// TwinCAT 3 PLC project plc
// ProgramVersion: 3.1.4024.0
// libraries:
//   Tc2_Standard, * (Beckhoff Automation GmbH)
//   Tc2_System, * (Beckhoff Automation GmbH)
//   Tc3_Module, * (Beckhoff Automation GmbH)
// project tree:
//   DUTs/ Axis_Command.TcDUT, Axis_Status.TcDUT
//   / PlcTask.TcTTO
//   POUs/ MAIN.TcPOU
// real-time tasks:
//   TASK PlcTask: cycle T#1ms, priority 4, ADS port 350
//   TASK PlcTask1: cycle T#2ms, priority 6, ADS port 351
// I/O:
//   DEVICE Device 2 (EtherCAT), AmsNetId 169.254.115.184.3.1
//     Box 2 (EX1616DN) [EX1616DN]
//       modules: Module 1 (SX1616DN)
//     p1 [MCDLN35BE]
//     j1 [MDDLN55BE]
//     j2 [MDDLN55BE]
//     j3 [MDDLN55BE]
//     j4 [MCDLN35BE]
//     j5 [MCDLN35BE]
//     j6 [MBDLN25BE]
//   DEVICE Device 4 (EtherCAT) (disabled), AmsNetId 172.16.9.47.5.1
//     zhua1 [ZeroErr Driver]
//     zhua2 [ZeroErr Driver]
//     kuaisubanshou1 [ZeroErr Driver] (disabled)
//     kuaisubanshou2 [ZeroErr Driver] (disabled)
//     kuaisubanshouqianjin [ZeroErr Driver] (disabled)
//   DEVICE Device 1 (EtherCAT) (disabled), AmsNetId 172.16.9.47.2.1
//     Drive 5 (ZeroErr Driver) [ZeroErr Driver]
// variable links:
//   plc2/plc2 Instance <-> Device 1 (EtherCAT)/Drive 5 (ZeroErr Driver)
//     PlcTask Inputs/MAIN.TW_STATUS/POSITION <-> Transmit PDO mapping 2/Position actual value
//     PlcTask Inputs/MAIN.TW_STATUS/STATUS_WORD <-> Transmit PDO mapping 2/Status word
//     PlcTask Inputs/MAIN.TW_STATUS/TORQUE_VALUE <-> Transmit PDO mapping 2/Torque actual value
//     PlcTask Outputs/MAIN.TW_COMMAND/CONTROL_WORD <-> Receive PDO mapping 8/Controlword
//     PlcTask Outputs/MAIN.TW_COMMAND/MAX_MOTOR_SPEED <-> Receive PDO mapping 8/Max motor speed
//     PlcTask Outputs/MAIN.TW_COMMAND/MODE_OF_OPERATION <-> Receive PDO mapping 8/Modes of operation
//     PlcTask Outputs/MAIN.TW_COMMAND/TARGET_TORQUE <-> Receive PDO mapping 8/Target torque
//   plc2/plc2 Instance <-> Device 4 (EtherCAT)/kuaisubanshou1
//     PlcTask Inputs/MAIN.T_Axis_3_STATUS/POSITION <-> Transmit PDO mapping 2/Position actual value
//     PlcTask Inputs/MAIN.T_Axis_3_STATUS/STATUS_WORD <-> Transmit PDO mapping 2/Status word
//     PlcTask Inputs/MAIN.T_Axis_3_STATUS/TORQUE_VALUE <-> Transmit PDO mapping 2/Torque actual value
//     PlcTask Outputs/MAIN.T_Axis_3_COMMAND/CONTROL_WORD <-> Receive PDO mapping 8/Controlword
//     PlcTask Outputs/MAIN.T_Axis_3_COMMAND/MAX_MOTOR_SPEED <-> Receive PDO mapping 8/Max motor speed
//     PlcTask Outputs/MAIN.T_Axis_3_COMMAND/MODE_OF_OPERATION <-> Receive PDO mapping 8/Modes of operation
//     PlcTask Outputs/MAIN.T_Axis_3_COMMAND/TARGET_TORQUE <-> Receive PDO mapping 8/Target torque
//   plc2/plc2 Instance <-> Device 4 (EtherCAT)/kuaisubanshou2
//     PlcTask Inputs/MAIN.T_Axis_4_STATUS/POSITION <-> Transmit PDO mapping 2/Position actual value
//     PlcTask Inputs/MAIN.T_Axis_4_STATUS/STATUS_WORD <-> Transmit PDO mapping 2/Status word
//     PlcTask Inputs/MAIN.T_Axis_4_STATUS/TORQUE_VALUE <-> Transmit PDO mapping 2/Torque actual value
//     PlcTask Outputs/MAIN.T_Axis_4_COMMAND/CONTROL_WORD <-> Receive PDO mapping 8/Controlword
//     PlcTask Outputs/MAIN.T_Axis_4_COMMAND/MAX_MOTOR_SPEED <-> Receive PDO mapping 8/Max motor speed
//     PlcTask Outputs/MAIN.T_Axis_4_COMMAND/MODE_OF_OPERATION <-> Receive PDO mapping 8/Modes of operation
//     PlcTask Outputs/MAIN.T_Axis_4_COMMAND/TARGET_TORQUE <-> Receive PDO mapping 8/Target torque
//   plc2/plc2 Instance <-> Device 4 (EtherCAT)/kuaisubanshouqianjin
//     PlcTask Inputs/MAIN.P_Axis_1_STATUS/POSITION_VALUE <-> Transmit PDO mapping 0/Position actual value
//     PlcTask Inputs/MAIN.P_Axis_1_STATUS/STATUS_WORD <-> Transmit PDO mapping 0/Status word
//     PlcTask Outputs/MAIN.P_Axis_1_COMMAND/CONTROL_WORD <-> Receive PDO mapping 7/Control word
//     PlcTask Outputs/MAIN.P_Axis_1_COMMAND/MODE_OF_OPERATION <-> Receive PDO mapping 7/Mode of operation
//     PlcTask Outputs/MAIN.P_Axis_1_COMMAND/TARGET_POSITION <-> Receive PDO mapping 7/Target Position
//   plc2/plc2 Instance <-> Device 4 (EtherCAT)/zhua1
//     PlcTask Inputs/MAIN.T_Axis_1_STATUS/POSITION <-> Transmit PDO mapping 2/Position actual value
//     PlcTask Inputs/MAIN.T_Axis_1_STATUS/STATUS_WORD <-> Transmit PDO mapping 2/Status word
//     PlcTask Inputs/MAIN.T_Axis_1_STATUS/TORQUE_VALUE <-> Transmit PDO mapping 2/Torque actual value
//     PlcTask Outputs/MAIN.T_Axis_1_COMMAND/CONTROL_WORD <-> Receive PDO mapping 8/Controlword
//     PlcTask Outputs/MAIN.T_Axis_1_COMMAND/MAX_MOTOR_SPEED <-> Receive PDO mapping 8/Max motor speed
//     PlcTask Outputs/MAIN.T_Axis_1_COMMAND/MODE_OF_OPERATION <-> Receive PDO mapping 8/Modes of operation
//     PlcTask Outputs/MAIN.T_Axis_1_COMMAND/TARGET_TORQUE <-> Receive PDO mapping 8/Target torque
//   plc2/plc2 Instance <-> Device 4 (EtherCAT)/zhua2
//     PlcTask Inputs/MAIN.T_Axis_2_STATUS/POSITION <-> Transmit PDO mapping 2/Position actual value
//     PlcTask Inputs/MAIN.T_Axis_2_STATUS/STATUS_WORD <-> Transmit PDO mapping 2/Status word
//     PlcTask Inputs/MAIN.T_Axis_2_STATUS/TORQUE_VALUE <-> Transmit PDO mapping 2/Torque actual value
//     PlcTask Outputs/MAIN.T_Axis_2_COMMAND/CONTROL_WORD <-> Receive PDO mapping 8/Controlword
//     PlcTask Outputs/MAIN.T_Axis_2_COMMAND/MAX_MOTOR_SPEED <-> Receive PDO mapping 8/Max motor speed
//     PlcTask Outputs/MAIN.T_Axis_2_COMMAND/MODE_OF_OPERATION <-> Receive PDO mapping 8/Modes of operation
//     PlcTask Outputs/MAIN.T_Axis_2_COMMAND/TARGET_TORQUE <-> Receive PDO mapping 8/Target torque
//   plc/plc Instance <-> Device 2 (EtherCAT)/Box 2 (EX1616DN)
//     PlcTask Outputs/MAIN.BREAK <-> Module 1 (SX1616DN)/Outputs/Digital16 OUT
//   plc/plc Instance <-> Device 2 (EtherCAT)/j1
//     PlcTask Inputs/MAIN.j1_status/Actual_Position <-> Transmit PDO mapping 1/Position actual value
//     PlcTask Inputs/MAIN.j1_status/Actual_Torque <-> Transmit PDO mapping 1/Torque actual value
//     PlcTask Inputs/MAIN.j1_status/Actual_Velocity <-> Transmit PDO mapping 1/Velocity actual value
//     PlcTask Inputs/MAIN.j1_status/Following_Err <-> Transmit PDO mapping 1/Following error actual value
//     PlcTask Inputs/MAIN.j1_status/Mode_of_Operation_disp <-> Transmit PDO mapping 1/Modes of operation display
//     PlcTask Inputs/MAIN.j1_status/status <-> Transmit PDO mapping 1/Statusword
//     PlcTask Outputs/MAIN.j1_acc <-> Receive PDO mapping 1/Profile acceleration
//     PlcTask Outputs/MAIN.j1_command/Control_Word <-> Receive PDO mapping 1/Controlword
//     PlcTask Outputs/MAIN.j1_command/Max_Motor_Speed <-> Receive PDO mapping 1/Max motor speed
//     PlcTask Outputs/MAIN.j1_command/Max_Torque <-> Receive PDO mapping 1/Max torque
//     PlcTask Outputs/MAIN.j1_command/Mode_of_Operation <-> Receive PDO mapping 1/Modes of operation
//     PlcTask Outputs/MAIN.j1_command/Profile_Velocity <-> Receive PDO mapping 1/Profile velocity
//     PlcTask Outputs/MAIN.j1_command/Target_Position <-> Receive PDO mapping 1/Target position
//     PlcTask Outputs/MAIN.j1_command/Target_Torque <-> Receive PDO mapping 1/Target torque
//     PlcTask Outputs/MAIN.j1_dacc <-> Receive PDO mapping 1/Profile deceleration
//   plc/plc Instance <-> Device 2 (EtherCAT)/j2
//     PlcTask Inputs/MAIN.j2_status/Actual_Position <-> Transmit PDO mapping 1/Position actual value
//     PlcTask Inputs/MAIN.j2_status/Actual_Torque <-> Transmit PDO mapping 1/Torque actual value
//     PlcTask Inputs/MAIN.j2_status/Actual_Velocity <-> Transmit PDO mapping 1/Velocity actual value
//     PlcTask Inputs/MAIN.j2_status/Following_Err <-> Transmit PDO mapping 1/Following error actual value
//     PlcTask Inputs/MAIN.j2_status/Mode_of_Operation_disp <-> Transmit PDO mapping 1/Modes of operation display
//     PlcTask Inputs/MAIN.j2_status/status <-> Transmit PDO mapping 1/Statusword
//     PlcTask Outputs/MAIN.j2_acc <-> Receive PDO mapping 1/Profile acceleration
//     PlcTask Outputs/MAIN.j2_command/Control_Word <-> Receive PDO mapping 1/Controlword
//     PlcTask Outputs/MAIN.j2_command/Max_Motor_Speed <-> Receive PDO mapping 1/Max motor speed
//     PlcTask Outputs/MAIN.j2_command/Max_Torque <-> Receive PDO mapping 1/Max torque
//     PlcTask Outputs/MAIN.j2_command/Mode_of_Operation <-> Receive PDO mapping 1/Modes of operation
//     PlcTask Outputs/MAIN.j2_command/Profile_Velocity <-> Receive PDO mapping 1/Profile velocity
//     PlcTask Outputs/MAIN.j2_command/Target_Position <-> Receive PDO mapping 1/Target position
//     PlcTask Outputs/MAIN.j2_command/Target_Torque <-> Receive PDO mapping 1/Target torque
//     PlcTask Outputs/MAIN.j2_dacc <-> Receive PDO mapping 1/Profile deceleration
//   plc/plc Instance <-> Device 2 (EtherCAT)/j3
//     PlcTask Inputs/MAIN.j3_status/Actual_Position <-> Transmit PDO mapping 1/Position actual value
//     PlcTask Inputs/MAIN.j3_status/Actual_Torque <-> Transmit PDO mapping 1/Torque actual value
//     PlcTask Inputs/MAIN.j3_status/Actual_Velocity <-> Transmit PDO mapping 1/Velocity actual value
//     PlcTask Inputs/MAIN.j3_status/Following_Err <-> Transmit PDO mapping 1/Following error actual value
//     PlcTask Inputs/MAIN.j3_status/Mode_of_Operation_disp <-> Transmit PDO mapping 1/Modes of operation display
//     PlcTask Inputs/MAIN.j3_status/status <-> Transmit PDO mapping 1/Statusword
//     PlcTask Outputs/MAIN.j3_acc <-> Receive PDO mapping 1/Profile acceleration
//     PlcTask Outputs/MAIN.j3_command/Control_Word <-> Receive PDO mapping 1/Controlword
//     PlcTask Outputs/MAIN.j3_command/Max_Motor_Speed <-> Receive PDO mapping 1/Max motor speed
//     PlcTask Outputs/MAIN.j3_command/Max_Torque <-> Receive PDO mapping 1/Max torque
//     PlcTask Outputs/MAIN.j3_command/Mode_of_Operation <-> Receive PDO mapping 1/Modes of operation
//     PlcTask Outputs/MAIN.j3_command/Profile_Velocity <-> Receive PDO mapping 1/Profile velocity
//     PlcTask Outputs/MAIN.j3_command/Target_Position <-> Receive PDO mapping 1/Target position
//     PlcTask Outputs/MAIN.j3_command/Target_Torque <-> Receive PDO mapping 1/Target torque
//     PlcTask Outputs/MAIN.j3_dacc <-> Receive PDO mapping 1/Profile deceleration
//   plc/plc Instance <-> Device 2 (EtherCAT)/j4
//     PlcTask Inputs/MAIN.j4_status/Actual_Position <-> Transmit PDO mapping 1/Position actual value
//     PlcTask Inputs/MAIN.j4_status/Actual_Torque <-> Transmit PDO mapping 1/Torque actual value
//     PlcTask Inputs/MAIN.j4_status/Actual_Velocity <-> Transmit PDO mapping 1/Velocity actual value
//     PlcTask Inputs/MAIN.j4_status/Following_Err <-> Transmit PDO mapping 1/Following error actual value
//     PlcTask Inputs/MAIN.j4_status/Mode_of_Operation_disp <-> Transmit PDO mapping 1/Modes of operation display
//     PlcTask Inputs/MAIN.j4_status/status <-> Transmit PDO mapping 1/Statusword
//     PlcTask Outputs/MAIN.j4_acc <-> Receive PDO mapping 1/Profile acceleration
//     PlcTask Outputs/MAIN.j4_command/Control_Word <-> Receive PDO mapping 1/Controlword
//     PlcTask Outputs/MAIN.j4_command/Max_Motor_Speed <-> Receive PDO mapping 1/Max motor speed
//     PlcTask Outputs/MAIN.j4_command/Max_Torque <-> Receive PDO mapping 1/Max torque
//     PlcTask Outputs/MAIN.j4_command/Mode_of_Operation <-> Receive PDO mapping 1/Modes of operation
//     PlcTask Outputs/MAIN.j4_command/Profile_Velocity <-> Receive PDO mapping 1/Profile velocity
//     PlcTask Outputs/MAIN.j4_command/Target_Position <-> Receive PDO mapping 1/Target position
//     PlcTask Outputs/MAIN.j4_command/Target_Torque <-> Receive PDO mapping 1/Target torque
//     PlcTask Outputs/MAIN.j4_dacc <-> Receive PDO mapping 1/Profile deceleration
//   plc/plc Instance <-> Device 2 (EtherCAT)/j5
//     PlcTask Inputs/MAIN.j5_status/Actual_Position <-> Transmit PDO mapping 1/Position actual value
//     PlcTask Inputs/MAIN.j5_status/Actual_Torque <-> Transmit PDO mapping 1/Torque actual value
//     PlcTask Inputs/MAIN.j5_status/Actual_Velocity <-> Transmit PDO mapping 1/Velocity actual value
//     PlcTask Inputs/MAIN.j5_status/Following_Err <-> Transmit PDO mapping 1/Following error actual value
//     PlcTask Inputs/MAIN.j5_status/Mode_of_Operation_disp <-> Transmit PDO mapping 1/Modes of operation display
//     PlcTask Inputs/MAIN.j5_status/status <-> Transmit PDO mapping 1/Statusword
//     PlcTask Outputs/MAIN.j5_acc <-> Receive PDO mapping 1/Profile acceleration
//     PlcTask Outputs/MAIN.j5_command/Control_Word <-> Receive PDO mapping 1/Controlword
//     PlcTask Outputs/MAIN.j5_command/Max_Motor_Speed <-> Receive PDO mapping 1/Max motor speed
//     PlcTask Outputs/MAIN.j5_command/Max_Torque <-> Receive PDO mapping 1/Max torque
//     PlcTask Outputs/MAIN.j5_command/Mode_of_Operation <-> Receive PDO mapping 1/Modes of operation
//     PlcTask Outputs/MAIN.j5_command/Profile_Velocity <-> Receive PDO mapping 1/Profile velocity
//     PlcTask Outputs/MAIN.j5_command/Target_Position <-> Receive PDO mapping 1/Target position
//     PlcTask Outputs/MAIN.j5_command/Target_Torque <-> Receive PDO mapping 1/Target torque
//     PlcTask Outputs/MAIN.j5_dacc <-> Receive PDO mapping 1/Profile deceleration
//   plc/plc Instance <-> Device 2 (EtherCAT)/j6
//     PlcTask Inputs/MAIN.j6_status/Actual_Position <-> Transmit PDO mapping 1/Position actual value
//     PlcTask Inputs/MAIN.j6_status/Actual_Torque <-> Transmit PDO mapping 1/Torque actual value
//     PlcTask Inputs/MAIN.j6_status/Actual_Velocity <-> Transmit PDO mapping 1/Velocity actual value
//     PlcTask Inputs/MAIN.j6_status/Following_Err <-> Transmit PDO mapping 1/Following error actual value
//     PlcTask Inputs/MAIN.j6_status/Mode_of_Operation_disp <-> Transmit PDO mapping 1/Modes of operation display
//     PlcTask Inputs/MAIN.j6_status/status <-> Transmit PDO mapping 1/Statusword
//     PlcTask Outputs/MAIN.j6_acc <-> Receive PDO mapping 1/Profile acceleration
//     PlcTask Outputs/MAIN.j6_command/Control_Word <-> Receive PDO mapping 1/Controlword
//     PlcTask Outputs/MAIN.j6_command/Max_Motor_Speed <-> Receive PDO mapping 1/Max motor speed
//     PlcTask Outputs/MAIN.j6_command/Max_Torque <-> Receive PDO mapping 1/Max torque
//     PlcTask Outputs/MAIN.j6_command/Mode_of_Operation <-> Receive PDO mapping 1/Modes of operation
//     PlcTask Outputs/MAIN.j6_command/Profile_Velocity <-> Receive PDO mapping 1/Profile velocity
//     PlcTask Outputs/MAIN.j6_command/Target_Position <-> Receive PDO mapping 1/Target position
//     PlcTask Outputs/MAIN.j6_command/Target_Torque <-> Receive PDO mapping 1/Target torque
//     PlcTask Outputs/MAIN.j6_dacc <-> Receive PDO mapping 1/Profile deceleration
//   plc/plc Instance <-> Device 2 (EtherCAT)/p1
//     PlcTask Inputs/MAIN.p1_status/Actual_Position <-> Transmit PDO mapping 1/Position actual value
//     PlcTask Inputs/MAIN.p1_status/Actual_Torque <-> Transmit PDO mapping 1/Torque actual value
//     PlcTask Inputs/MAIN.p1_status/Actual_Velocity <-> Transmit PDO mapping 1/Velocity actual value
//     PlcTask Inputs/MAIN.p1_status/Following_Err <-> Transmit PDO mapping 1/Following error actual value
//     PlcTask Inputs/MAIN.p1_status/Mode_of_Operation_disp <-> Transmit PDO mapping 1/Modes of operation display
//     PlcTask Inputs/MAIN.p1_status/status <-> Transmit PDO mapping 1/Statusword
//     PlcTask Outputs/MAIN.p1_command/Control_Word <-> Receive PDO mapping 1/Controlword
//     PlcTask Outputs/MAIN.p1_command/Max_Motor_Speed <-> Receive PDO mapping 1/Max motor speed
//     PlcTask Outputs/MAIN.p1_command/Max_Torque <-> Receive PDO mapping 1/Max torque
//     PlcTask Outputs/MAIN.p1_command/Mode_of_Operation <-> Receive PDO mapping 1/Modes of operation
//     PlcTask Outputs/MAIN.p1_command/Profile_Velocity <-> Receive PDO mapping 1/Profile velocity
//     PlcTask Outputs/MAIN.p1_command/Target_Position <-> Receive PDO mapping 1/Target position
//     PlcTask Outputs/MAIN.p1_command/Target_Torque <-> Receive PDO mapping 1/Target torque
//     PlcTask Outputs/MAIN.q1_acc <-> Receive PDO mapping 1/Profile acceleration
//     PlcTask Outputs/MAIN.q1_dacc <-> Receive PDO mapping 1/Profile deceleration

CONFIGURATION plc
    RESOURCE PLC ON TwinCAT3
        TASK PlcTask(INTERVAL := T#1ms, PRIORITY := 4);
        PROGRAM MAIN WITH PlcTask : MAIN;
    END_RESOURCE
END_CONFIGURATION

// ---- DUTs/Axis_Command.TcDUT
TYPE Axis_Command :
STRUCT
	Control_Word AT%Q* :WORD;
	Target_Position AT%Q* :DINT;
	Profile_Velocity AT%Q*:UDINT;
	Max_Motor_Speed AT%Q* :UDINT;
	Mode_of_Operation AT%Q* :BYTE:=1;
	Target_Torque AT%Q*: INT:=0;
	Max_Torque AT%Q*: UINT:=0;
END_STRUCT
END_TYPE

// ---- DUTs/Axis_Status.TcDUT
TYPE Axis_Status :
STRUCT
	status: WORD;
	Mode_of_Operation_disp :BYTE;
	Actual_Position:DINT;
	Actual_Velocity:DINT;
	Following_Err : DINT;
	Actual_Torque:INT;
END_STRUCT
END_TYPE

// ---- POUs/MAIN.TcPOU
PROGRAM MAIN
VAR
	j1_command AT%QD0:Axis_Command;
	j2_command AT%QD6:Axis_Command;
	j3_command AT%QD12:Axis_Command;
	j4_command AT%QD18:Axis_Command;
	j5_command AT%QD24:Axis_Command;
	j6_command AT%QD30:Axis_Command;
	p1_command AT%QD36:Axis_Command;
	
	j1_status AT%ID0:Axis_Status;
	j2_status AT%ID5:Axis_Status;
	j3_status AT%ID10:Axis_Status;
	j4_status AT%ID15:Axis_Status;
	j5_status AT%ID20:Axis_Status;
	j6_status AT%ID25:Axis_Status;
	p1_status AT%ID30:Axis_Status;
	
	BREAK AT%QD100:WORD:=8;
	
	j1_acc AT%Q*:UDINT :=40000000;
	j2_acc AT%Q*:UDINT :=40000000;
	j3_acc AT%Q*:UDINT :=40000000;
	j4_acc AT%Q*:UDINT :=4000000000;
	j5_acc AT%Q*:UDINT :=40000000;
	j6_acc AT%Q*:UDINT :=40000000;
	j1_dacc AT%Q*:UDINT :=40000000;
	j2_dacc AT%Q*:UDINT :=40000000;
	j3_dacc AT%Q*:UDINT :=40000000;
	j4_dacc AT%Q*:UDINT :=4000000000;
	j5_dacc AT%Q*:UDINT :=40000000;
	j6_dacc AT%Q*:UDINT :=40000000;
	q1_acc AT%Q*:UDINT :=40000000;
	q1_dacc AT%Q*:UDINT :=400000000;
	
	tool_sensor AT%ID100:INT;
END_VAR

END_PROGRAM
